{attribute addProperty BoxType "EL5042-0000-0016"}
{attribute addProperty Id "FB_Inputs_ChannelAT %I*ARRAY[0..2] OF FB_Inputs_Channel_FFB44ACB160200WcStateAT %I*WcState_98A4DF7520.250InfoDataAT %I*InfoData_BC63D37F80100"}
{attribute addProperty CRC "2346587001"}
{attribute addProperty SizeInBites "242"}
{attribute addProperty SizeInBytes "30.25"}
TYPE EL5042_3D8BD04C :
STRUCT
	{attribute addProperty Name "FB_Inputs_Channel"}
	FB_Inputs_Channel : ARRAY[0..2] OF FB_Inputs_Channel_FFB44ACB;
	{attribute addProperty Name "WcState"}
	WcState : WcState_98A4DF75;
	{attribute addProperty Name "InfoData"}
	InfoData : InfoData_BC63D37F;
END_STRUCT
END_TYPE

(* stored: Version 1.2.0.0, ProductVersion 3.1.4024.9
   DUT EL5042_3D8BD04C: Id {505430a3-13f1-4ae7-95b9-2fa64a4e1e34} *)
